Staubli VAL3: _toString.pgx

program _toString(string x_sRow, num x_nColumn, string& x_sString[])
begin
  x_sString=x_sRow+mid("000",3-len(toString("",x_nColumn)),0)+toString("",x_nColumn)
end
